# EPICS alarm handler configuration: mps_database/bare/alarms/areas/mpln_gunb_mp01.alhConfig
GROUP NULL MPLN:GUNB:MP01:1
$ALIAS MPS Link Node 50
$GUIDANCE
LTUH MPS
   Group Name: MPLN:GUNB:MP01:1
   Summary PV:  MPLN:GUNB:MP01:1:STATSUMY
$END
CHANNEL  MPLN:GUNB:MP01:1    MPLN:GUNB:MP01:1:MPS_EN_RBV		-----
CHANNEL  MPLN:GUNB:MP01:1    MPLN:GUNB:MP01:1:LC1_MODE_RBV		-----
